(* Logix 5000 project; controller EuniceF_ICA10 vendor 1 type 14 code 150 rev 37.11; software revision 37.00 *)

TASK MainTask (continuous, watchdog 500 ms) : MainProgram

MODULES
   Local : vendor 1 type 14 code 150 (Compact 0, rev 37.11)
      Analog_IO : Embedded (Compact 2, rev 1.1, Output RPI 80 ms)
      Discrete_IO : Embedded (Compact 1, rev 3.1, Output RPI 20 ms)
      Counters : Embedded (Compact 3, rev 1.1, Output RPI 20 ms)
END_MODULES

VAR_GLOBAL   (* controller tags *)
   ACCELERATE : ALIAS FOR Local:1:I.Data.11;
   ALERT : ALIAS FOR Local:1:O.Data.4;
   DECELERATE : ALIAS FOR Local:1:I.Data.12;
   M_ACCELERATE : ALIAS FOR Local:1:O.Data.1;
   M_DECELERATE : ALIAS FOR Local:1:O.Data.2;
   M_STOP : ALIAS FOR Local:1:O.Data.3;
   PRESENT : ALIAS FOR Local:1:I.Data.0;
   STOPPED : ALIAS FOR Local:1:I.Data.15;
   STOPPEDSWITCH : ALIAS FOR Local:1:I.Data.1;
   TIMEOUT : ALIAS FOR Local:1:O.Data.5;
   TIMER1 : TIMER := (PRE := 3000);
END_VAR

PROGRAM MainProgram   (* main routine MainRoutine *)

ROUTINE MainRoutine   (* ladder *)
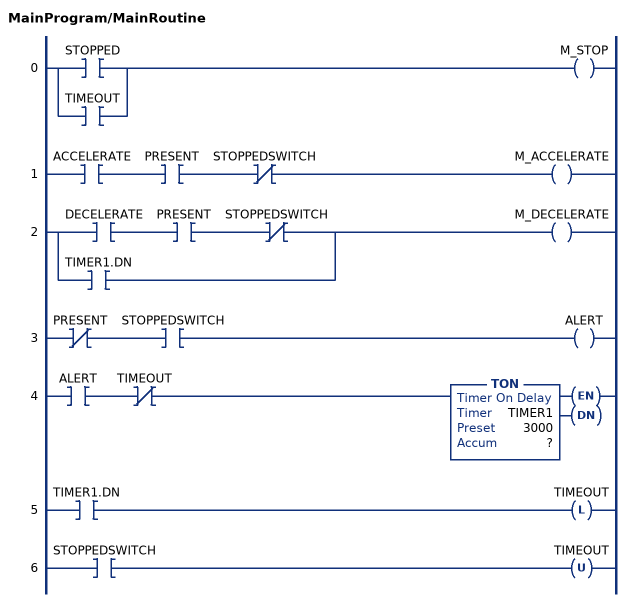
   0: [XIC(STOPPED) ,XIC(TIMEOUT) ]OTE(M_STOP);
   1: XIC(ACCELERATE)XIC(PRESENT)XIO(STOPPEDSWITCH)OTE(M_ACCELERATE);
   2: [XIC(DECELERATE) XIC(PRESENT) XIO(STOPPEDSWITCH) ,XIC(TIMER1.DN) ]OTE(M_DECELERATE);
   3: XIO(PRESENT)XIC(STOPPEDSWITCH)OTE(ALERT);
   4: XIC(ALERT)XIO(TIMEOUT)TON(TIMER1,?,?);
   5: XIC(TIMER1.DN)OTL(TIMEOUT);
   6: XIC(STOPPEDSWITCH)OTU(TIMEOUT);
END_ROUTINE
END_PROGRAM
